FUNCTION_BLOCK PUBLISH_1 (* Single-Variable Publisher *)
  (* Standard: 61499-1-3.2 *)
  (* Version 0.1, 2001-04-24, JHC, Rockwell Automation, XML version *)
  (* Version 0.0, 1998-12-08, JHC, Rockwell Automation, SRC version *)
  (* Compiler header: package fb.rt.net; *)
  (* Compiler Java IBM VisualAge 3.0 *)
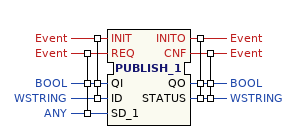
  EVENT_INPUT
    INIT WITH QI, ID; (* Service Initialization *)
    REQ WITH QI, SD_1; (* Service Request *)
  END_EVENT
  EVENT_OUTPUT
    INITO WITH QO, STATUS; (* Initialization Confirm *)
    CNF WITH QO, STATUS; (* Service Confirmation *)
  END_EVENT
  VAR_INPUT
    QI : BOOL; (* Event Input Qualifier *)
    ID : WSTRING; (* Connection Identifier *)
    SD_1 : ANY; (* Data to Send *)
  END_VAR
  VAR_OUTPUT
    QO : BOOL; (* Event Output Qualifier *)
    STATUS : WSTRING; (* Service Status *)
  END_VAR
  SERVICE PUBLISH_1/SUBSCRIBE_1 (* Data Publication Service *)
    SEQUENCE normal_establishment
      PUBLISH_1.INIT+(ID) -> PUBLISH_1.INITO+();
      SUBSCRIBE_1.INIT+(ID) -> SUBSCRIBE_1.INITO+();
    END_SEQUENCE
    SEQUENCE publisher_rejected_establishment
      PUBLISH_1.INIT+(ID) -> PUBLISH_1.INITO-(STATUS);
    END_SEQUENCE
    SEQUENCE subscriber_rejected_establishment
      SUBSCRIBE_1.INIT+(ID) -> SUBSCRIBE_1.INITO-(STATUS);
    END_SEQUENCE
    SEQUENCE normal_data_transfer
      PUBLISH_1.REQ+(SD_1) -> SUBSCRIBE_1.IND+(RD_1);
      -> PUBLISH_1.CNF+();
      SUBSCRIBE_1.RSP+();
    END_SEQUENCE
    SEQUENCE data_transfer_error
      PUBLISH_1.REQ+(SD_1) -> SUBSCRIBE_1.IND-(STATUS);
      -> PUBLISH_1.CNF+();
    END_SEQUENCE
    SEQUENCE publisher_initiated_disconnect
      PUBLISH_1.INIT-() -> SUBSCRIBE_1.INITO-(STATUS);
      -> PUBLISH_1.INITO-(STATUS);
    END_SEQUENCE
    SEQUENCE subscriber_initiated_disconnect
      SUBSCRIBE_1.INIT-() -> SUBSCRIBE_1.INITO-(STATUS);
    END_SEQUENCE
    SEQUENCE system_publisher_disconnect
      -> PUBLISH_1.INITO-(STATUS);
      -> SUBSCRIBE_1.INITO-(STATUS);
    END_SEQUENCE
    SEQUENCE system_subscriber_disconnect
      -> SUBSCRIBE_1.INITO-(STATUS);
    END_SEQUENCE
  END_SERVICE
END_FUNCTION_BLOCK
